% RSLogix 500 project Glycol_2.RSS, saved by version 12.00.00.00 %
PROJECT "GOODFOOD"    % processor: Bul.1763 MicroLogix 1100 Series B %

PROGRAM FILES
  LAD 2   24 rungs
  LAD 3   18 rungs
  LAD 4   25 rungs
  LAD 5   58 rungs

DATA FILES
  O0 OUTPUT  9 elements
  I1 INPUT  23 elements
  S2 STATUS  66 elements
  B3 BINARY  1 elements
  T4 TIMER  19 elements
  C5 COUNTER  9 elements
  R6 CONTROL  1 elements
  N7 INTEGER  11 elements
  F8 FLOAT  39 elements
  F9   45 elements
  B10   2 elements
  F11   14 elements
  F12   8 elements
  T13   7 elements
  F14   10 elements
  F15   10 elements
  B16   2 elements
  PD17   1 elements
  PD18   1 elements
  N19   23 elements
  F20   40 elements

LADDER 2
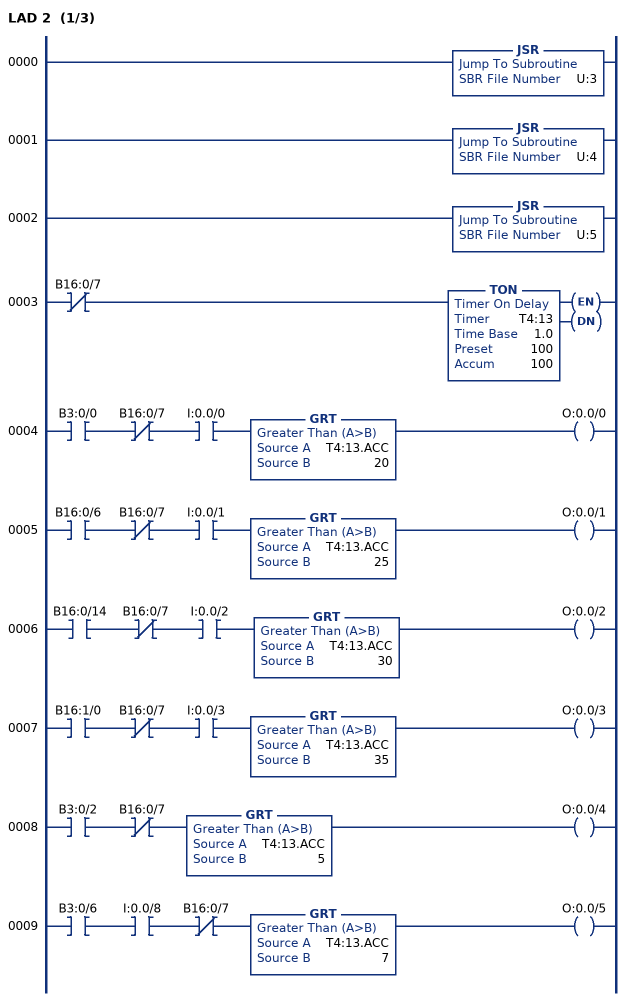
% Rung: 0 %
SOR JSR U:3 EOR
% Rung: 1 %
SOR JSR U:4 EOR
% Rung: 2 %
SOR JSR U:5 EOR
% Rung: 3 %
SOR XIO B16:0/7 TON T4:13 1.0 100 100 EOR
% Rung: 4 %
SOR XIC B3:0/0 XIO B16:0/7 XIC I:0.0/0 GRT T4:13.ACC 20 OTE O:0.0/0 EOR
% Rung: 5 %
SOR XIC B16:0/6 XIO B16:0/7 XIC I:0.0/1 GRT T4:13.ACC 25 OTE O:0.0/1 EOR
% Rung: 6 %
SOR XIC B16:0/14 XIO B16:0/7 XIC I:0.0/2 GRT T4:13.ACC 30 OTE O:0.0/2 EOR
% Rung: 7 %
SOR XIC B16:1/0 XIO B16:0/7 XIC I:0.0/3 GRT T4:13.ACC 35 OTE O:0.0/3 EOR
% Rung: 8 %
SOR XIC B3:0/2 XIO B16:0/7 GRT T4:13.ACC 5 OTE O:0.0/4 EOR
% Rung: 9 %
SOR XIC B3:0/6 XIC I:0.0/8 XIO B16:0/7 GRT T4:13.ACC 7 OTE O:0.0/5 EOR

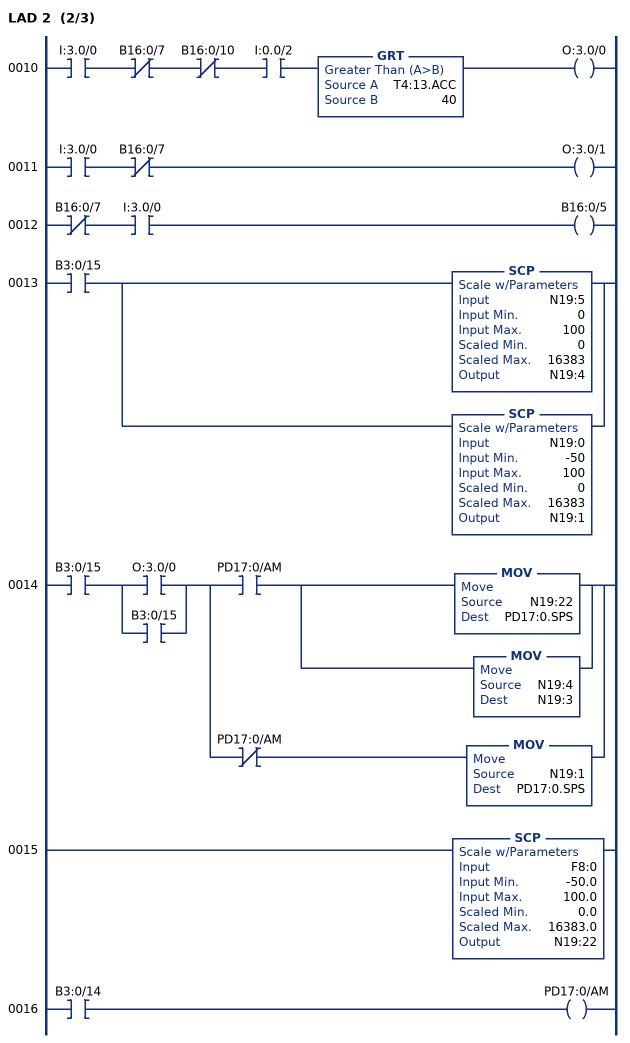
% Rung: 10 %
SOR XIC I:3.0/0 XIO B16:0/7 XIO B16:0/10 XIC I:0.0/2 GRT T4:13.ACC 40 OTE O:3.0/0 EOR
% Rung: 11 %
SOR XIC I:3.0/0 XIO B16:0/7 OTE O:3.0/1 EOR
% Rung: 12 %
SOR XIO B16:0/7 XIC I:3.0/0 OTE B16:0/5 EOR
% Rung: 13 %
SOR XIC B3:0/15 BST SCP N19:5 0 100 0 16383 N19:4 NXB SCP N19:0 -50 100 0 16383 N19:1 BND EOR
% Rung: 14 %
SOR XIC B3:0/15 BST XIC O:3.0/0 NXB XIC B3:0/15 BND BST XIC PD17:0/AM BST MOV N19:22 PD17:0.SPS NXB MOV N19:4 N19:3 BND NXB XIO PD17:0/AM MOV N19:1 PD17:0.SPS BND EOR
% Rung: 15 %
SOR SCP F8:0 -50.0 100.0 0.0 16383.0 N19:22 EOR
% Rung: 16 %
SOR XIC B3:0/14 OTE PD17:0/AM EOR

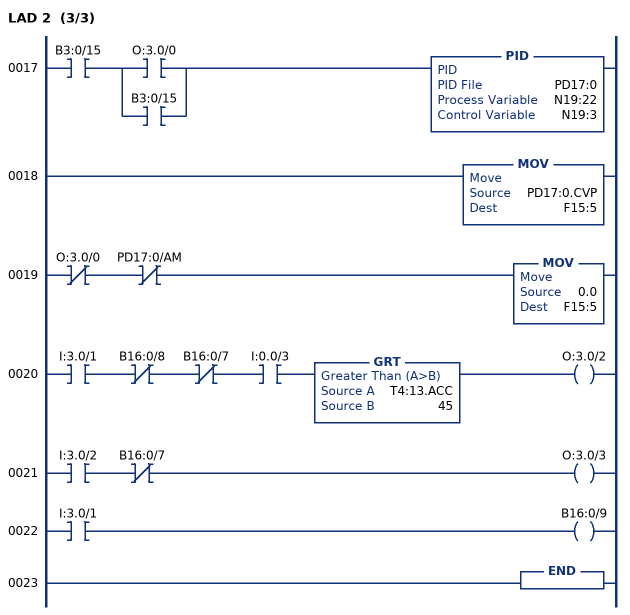
% Rung: 17 %
SOR XIC B3:0/15 BST XIC O:3.0/0 NXB XIC B3:0/15 BND PID PD17:0 N19:22 N19:3 EOR
% Rung: 18 %
SOR MOV PD17:0.CVP F15:5 EOR
% Rung: 19 %
SOR XIO O:3.0/0 XIO PD17:0/AM MOV 0.0 F15:5 EOR
% Rung: 20 %
SOR XIC I:3.0/1 XIO B16:0/8 XIO B16:0/7 XIC I:0.0/3 GRT T4:13.ACC 45 OTE O:3.0/2 EOR
% Rung: 21 %
SOR XIC I:3.0/2 XIO B16:0/7 OTE O:3.0/3 EOR
% Rung: 22 %
SOR XIC I:3.0/1 OTE B16:0/9 EOR
% Rung: 23 %
SOR END EOR

LADDER 3
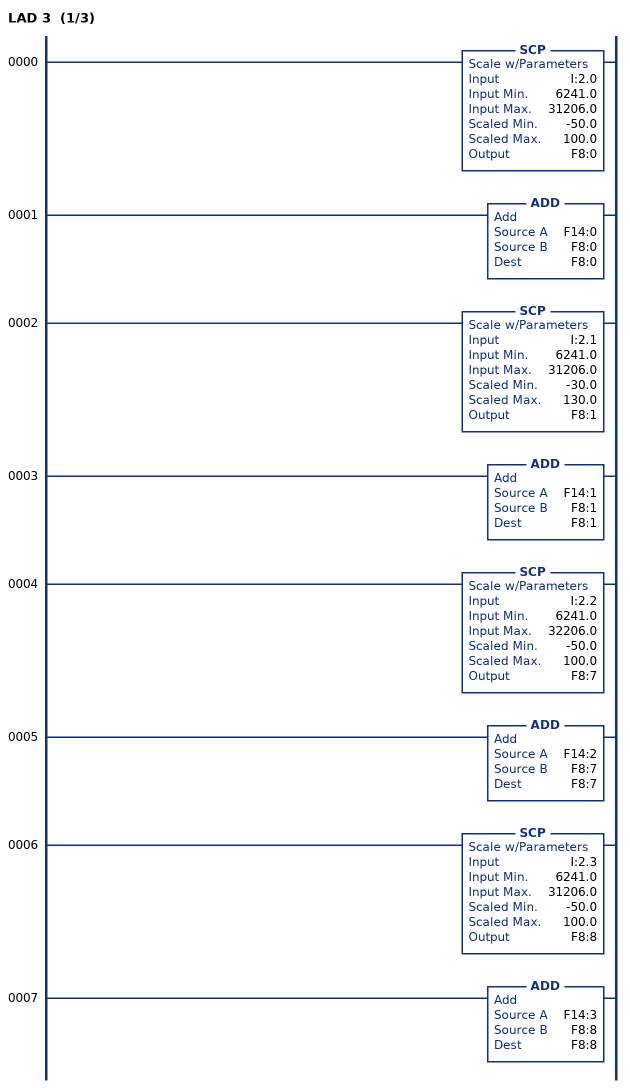
% Rung: 0 %
SOR SCP I:2.0 6241.0 31206.0 -50.0 100.0 F8:0 EOR
% Rung: 1 %
SOR ADD F14:0 F8:0 F8:0 EOR
% Rung: 2 %
SOR SCP I:2.1 6241.0 31206.0 -30.0 130.0 F8:1 EOR
% Rung: 3 %
SOR ADD F14:1 F8:1 F8:1 EOR
% Rung: 4 %
SOR SCP I:2.2 6241.0 32206.0 -50.0 100.0 F8:7 EOR
% Rung: 5 %
SOR ADD F14:2 F8:7 F8:7 EOR
% Rung: 6 %
SOR SCP I:2.3 6241.0 31206.0 -50.0 100.0 F8:8 EOR
% Rung: 7 %
SOR ADD F14:3 F8:8 F8:8 EOR

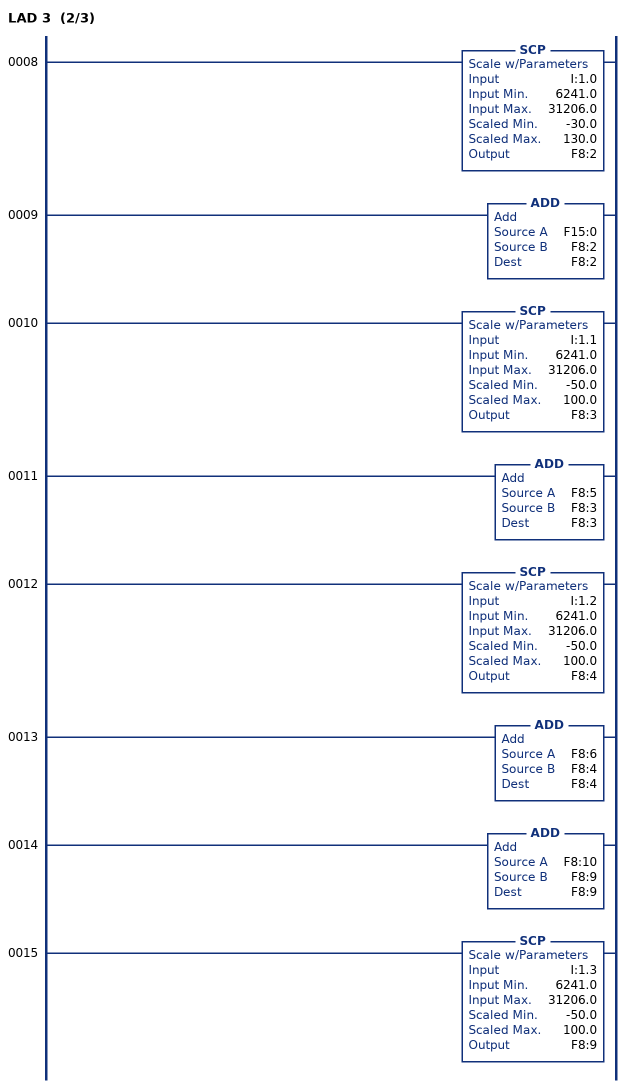
% Rung: 8 %
SOR SCP I:1.0 6241.0 31206.0 -30.0 130.0 F8:2 EOR
% Rung: 9 %
SOR ADD F15:0 F8:2 F8:2 EOR
% Rung: 10 %
SOR SCP I:1.1 6241.0 31206.0 -50.0 100.0 F8:3 EOR
% Rung: 11 %
SOR ADD F8:5 F8:3 F8:3 EOR
% Rung: 12 %
SOR SCP I:1.2 6241.0 31206.0 -50.0 100.0 F8:4 EOR
% Rung: 13 %
SOR ADD F8:6 F8:4 F8:4 EOR
% Rung: 14 %
SOR ADD F8:10 F8:9 F8:9 EOR
% Rung: 15 %
SOR SCP I:1.3 6241.0 31206.0 -50.0 100.0 F8:9 EOR

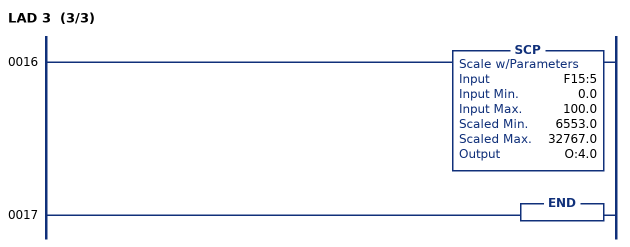
% Rung: 16 %
SOR SCP F15:5 0.0 100.0 6553.0 32767.0 O:4.0 EOR
% Rung: 17 %
SOR END EOR

LADDER 4
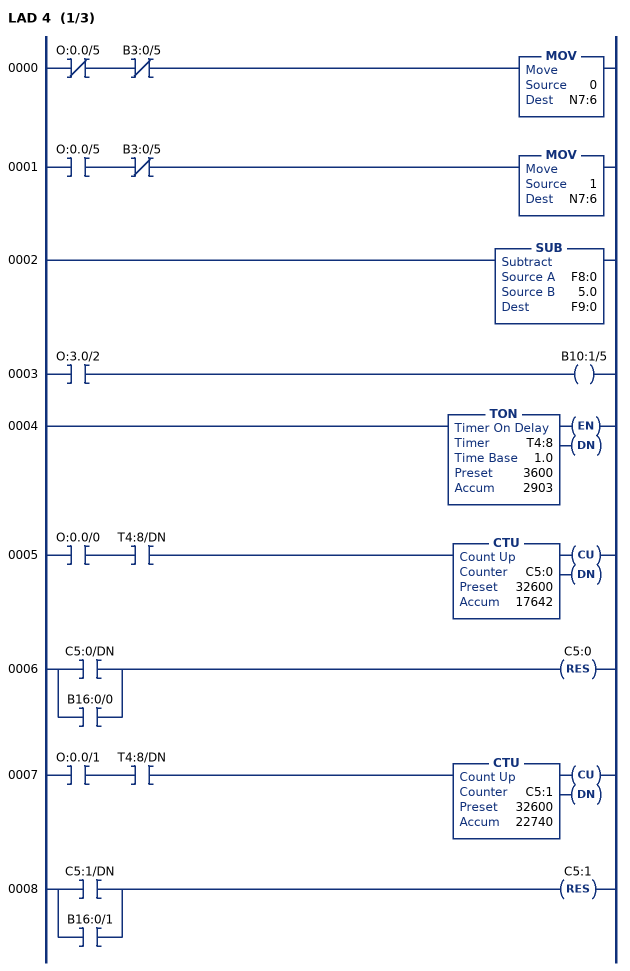
% Rung: 0 %
SOR XIO O:0.0/5 XIO B3:0/5 MOV 0 N7:6 EOR
% Rung: 1 %
SOR XIC O:0.0/5 XIO B3:0/5 MOV 1 N7:6 EOR
% Rung: 2 %
SOR SUB F8:0 5.0 F9:0 EOR
% Rung: 3 %
SOR XIC O:3.0/2 OTE B10:1/5 EOR
% Rung: 4 %
SOR TON T4:8 1.0 3600 2903 EOR
% Rung: 5 %
SOR XIC O:0.0/0 XIC T4:8/DN CTU C5:0 32600 17642 EOR
% Rung: 6 %
SOR BST XIC C5:0/DN NXB XIC B16:0/0 BND RES C5:0 EOR
% Rung: 7 %
SOR XIC O:0.0/1 XIC T4:8/DN CTU C5:1 32600 22740 EOR
% Rung: 8 %
SOR BST XIC C5:1/DN NXB XIC B16:0/1 BND RES C5:1 EOR

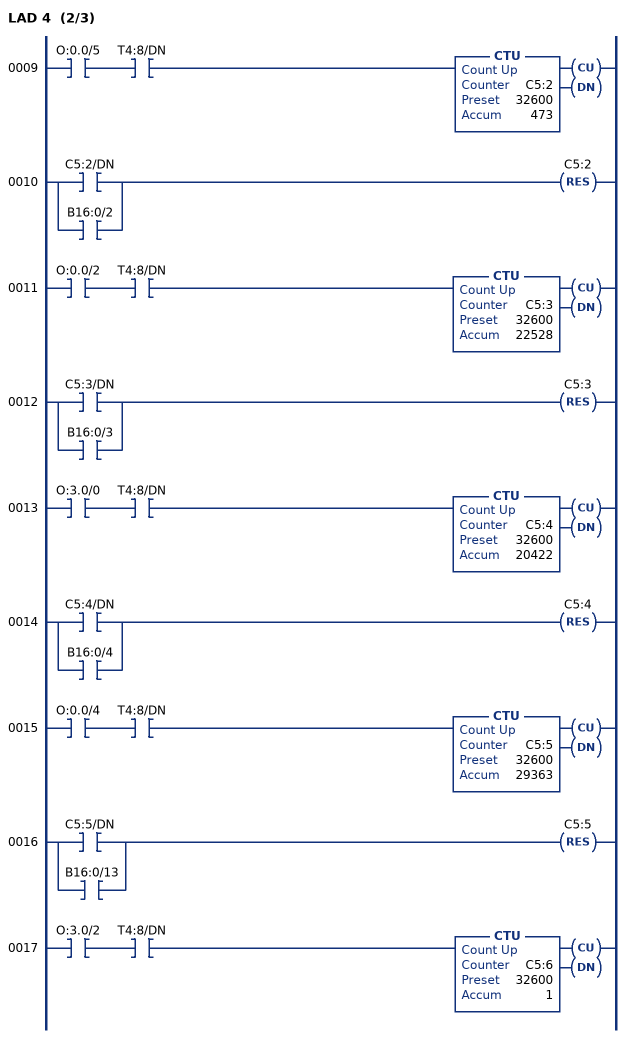
% Rung: 9 %
SOR XIC O:0.0/5 XIC T4:8/DN CTU C5:2 32600 473 EOR
% Rung: 10 %
SOR BST XIC C5:2/DN NXB XIC B16:0/2 BND RES C5:2 EOR
% Rung: 11 %
SOR XIC O:0.0/2 XIC T4:8/DN CTU C5:3 32600 22528 EOR
% Rung: 12 %
SOR BST XIC C5:3/DN NXB XIC B16:0/3 BND RES C5:3 EOR
% Rung: 13 %
SOR XIC O:3.0/0 XIC T4:8/DN CTU C5:4 32600 20422 EOR
% Rung: 14 %
SOR BST XIC C5:4/DN NXB XIC B16:0/4 BND RES C5:4 EOR
% Rung: 15 %
SOR XIC O:0.0/4 XIC T4:8/DN CTU C5:5 32600 29363 EOR
% Rung: 16 %
SOR BST XIC C5:5/DN NXB XIC B16:0/13 BND RES C5:5 EOR
% Rung: 17 %
SOR XIC O:3.0/2 XIC T4:8/DN CTU C5:6 32600 1 EOR

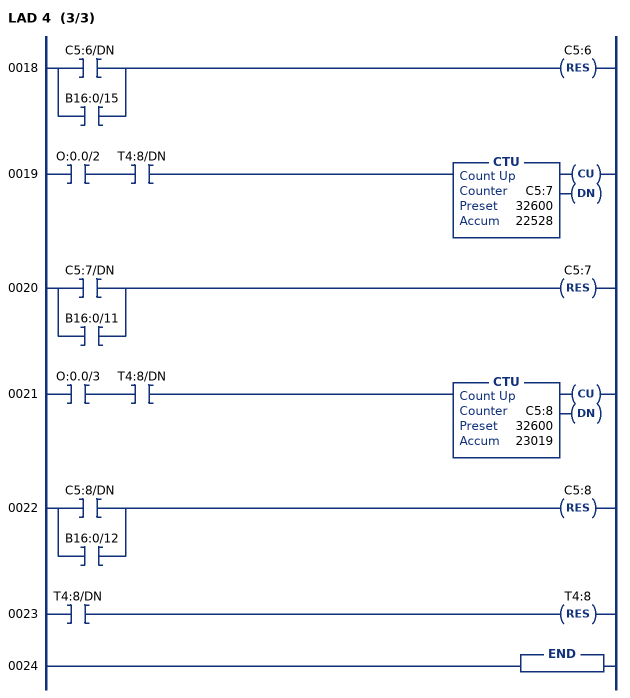
% Rung: 18 %
SOR BST XIC C5:6/DN NXB XIC B16:0/15 BND RES C5:6 EOR
% Rung: 19 %
SOR XIC O:0.0/2 XIC T4:8/DN CTU C5:7 32600 22528 EOR
% Rung: 20 %
SOR BST XIC C5:7/DN NXB XIC B16:0/11 BND RES C5:7 EOR
% Rung: 21 %
SOR XIC O:0.0/3 XIC T4:8/DN CTU C5:8 32600 23019 EOR
% Rung: 22 %
SOR BST XIC C5:8/DN NXB XIC B16:0/12 BND RES C5:8 EOR
% Rung: 23 %
SOR XIC T4:8/DN RES T4:8 EOR
% Rung: 24 %
SOR END EOR

LADDER 5
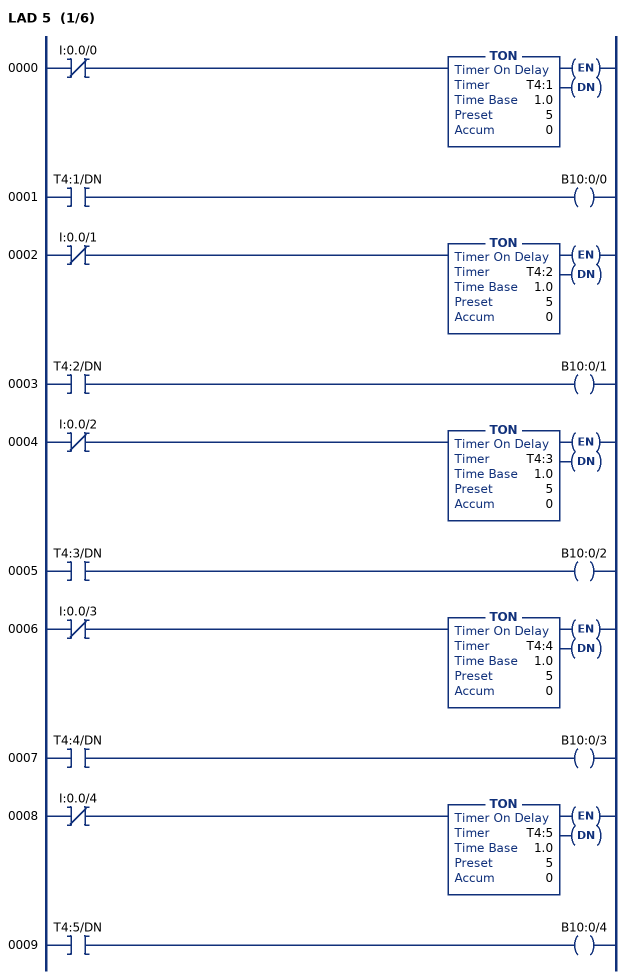
% Rung: 0 %
SOR XIO I:0.0/0 TON T4:1 1.0 5 0 EOR
% Rung: 1 %
SOR XIC T4:1/DN OTE B10:0/0 EOR
% Rung: 2 %
SOR XIO I:0.0/1 TON T4:2 1.0 5 0 EOR
% Rung: 3 %
SOR XIC T4:2/DN OTE B10:0/1 EOR
% Rung: 4 %
SOR XIO I:0.0/2 TON T4:3 1.0 5 0 EOR
% Rung: 5 %
SOR XIC T4:3/DN OTE B10:0/2 EOR
% Rung: 6 %
SOR XIO I:0.0/3 TON T4:4 1.0 5 0 EOR
% Rung: 7 %
SOR XIC T4:4/DN OTE B10:0/3 EOR
% Rung: 8 %
SOR XIO I:0.0/4 TON T4:5 1.0 5 0 EOR
% Rung: 9 %
SOR XIC T4:5/DN OTE B10:0/4 EOR

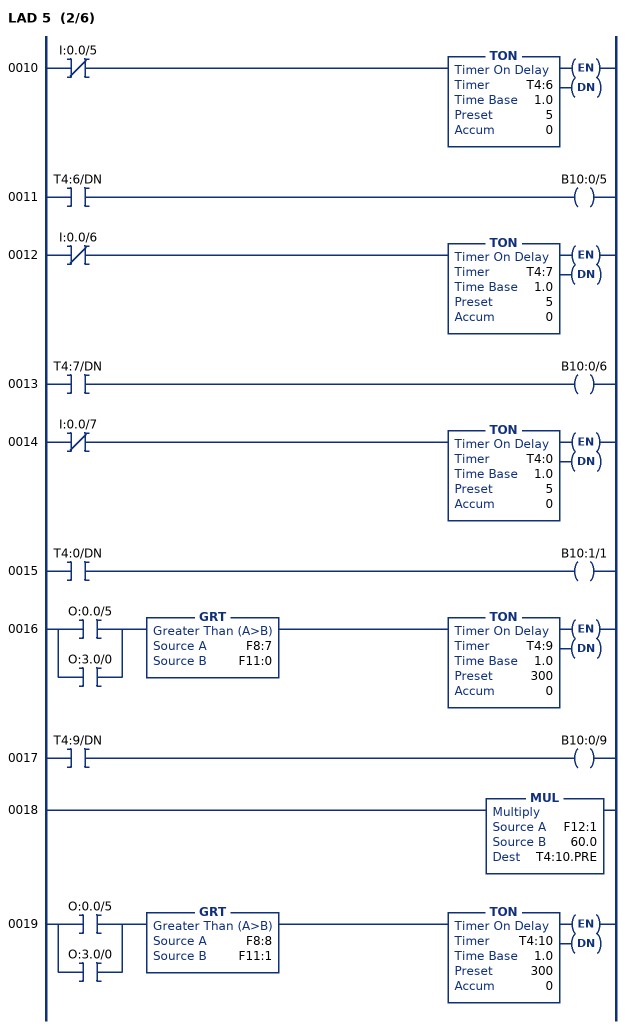
% Rung: 10 %
SOR XIO I:0.0/5 TON T4:6 1.0 5 0 EOR
% Rung: 11 %
SOR XIC T4:6/DN OTE B10:0/5 EOR
% Rung: 12 %
SOR XIO I:0.0/6 TON T4:7 1.0 5 0 EOR
% Rung: 13 %
SOR XIC T4:7/DN OTE B10:0/6 EOR
% Rung: 14 %
SOR XIO I:0.0/7 TON T4:0 1.0 5 0 EOR
% Rung: 15 %
SOR XIC T4:0/DN OTE B10:1/1 EOR
% Rung: 16 %
SOR BST XIC O:0.0/5 NXB XIC O:3.0/0 BND GRT F8:7 F11:0 TON T4:9 1.0 300 0 EOR
% Rung: 17 %
SOR XIC T4:9/DN OTE B10:0/9 EOR
% Rung: 18 %
SOR MUL F12:1 60.0 T4:10.PRE EOR
% Rung: 19 %
SOR BST XIC O:0.0/5 NXB XIC O:3.0/0 BND GRT F8:8 F11:1 TON T4:10 1.0 300 0 EOR

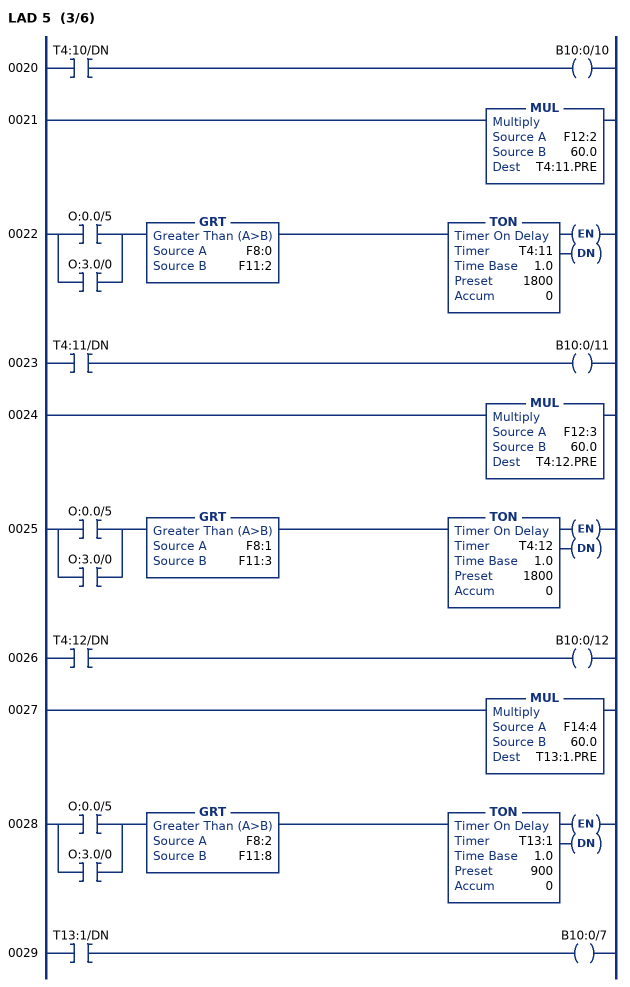
% Rung: 20 %
SOR XIC T4:10/DN OTE B10:0/10 EOR
% Rung: 21 %
SOR MUL F12:2 60.0 T4:11.PRE EOR
% Rung: 22 %
SOR BST XIC O:0.0/5 NXB XIC O:3.0/0 BND GRT F8:0 F11:2 TON T4:11 1.0 1800 0 EOR
% Rung: 23 %
SOR XIC T4:11/DN OTE B10:0/11 EOR
% Rung: 24 %
SOR MUL F12:3 60.0 T4:12.PRE EOR
% Rung: 25 %
SOR BST XIC O:0.0/5 NXB XIC O:3.0/0 BND GRT F8:1 F11:3 TON T4:12 1.0 1800 0 EOR
% Rung: 26 %
SOR XIC T4:12/DN OTE B10:0/12 EOR
% Rung: 27 %
SOR MUL F14:4 60.0 T13:1.PRE EOR
% Rung: 28 %
SOR BST XIC O:0.0/5 NXB XIC O:3.0/0 BND GRT F8:2 F11:8 TON T13:1 1.0 900 0 EOR
% Rung: 29 %
SOR XIC T13:1/DN OTE B10:0/7 EOR

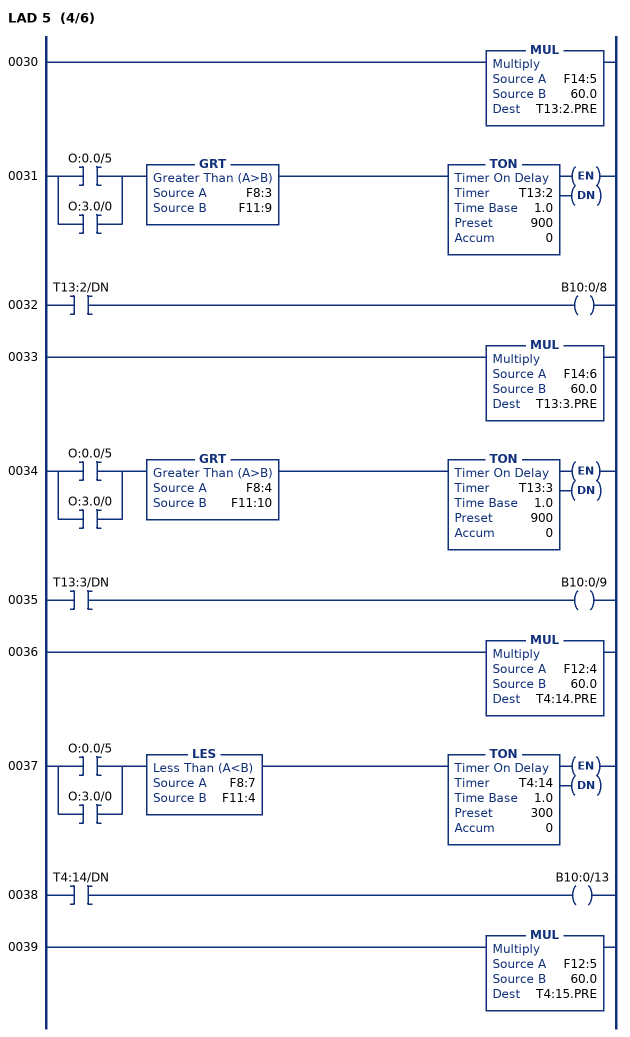
% Rung: 30 %
SOR MUL F14:5 60.0 T13:2.PRE EOR
% Rung: 31 %
SOR BST XIC O:0.0/5 NXB XIC O:3.0/0 BND GRT F8:3 F11:9 TON T13:2 1.0 900 0 EOR
% Rung: 32 %
SOR XIC T13:2/DN OTE B10:0/8 EOR
% Rung: 33 %
SOR MUL F14:6 60.0 T13:3.PRE EOR
% Rung: 34 %
SOR BST XIC O:0.0/5 NXB XIC O:3.0/0 BND GRT F8:4 F11:10 TON T13:3 1.0 900 0 EOR
% Rung: 35 %
SOR XIC T13:3/DN OTE B10:0/9 EOR
% Rung: 36 %
SOR MUL F12:4 60.0 T4:14.PRE EOR
% Rung: 37 %
SOR BST XIC O:0.0/5 NXB XIC O:3.0/0 BND LES F8:7 F11:4 TON T4:14 1.0 300 0 EOR
% Rung: 38 %
SOR XIC T4:14/DN OTE B10:0/13 EOR
% Rung: 39 %
SOR MUL F12:5 60.0 T4:15.PRE EOR

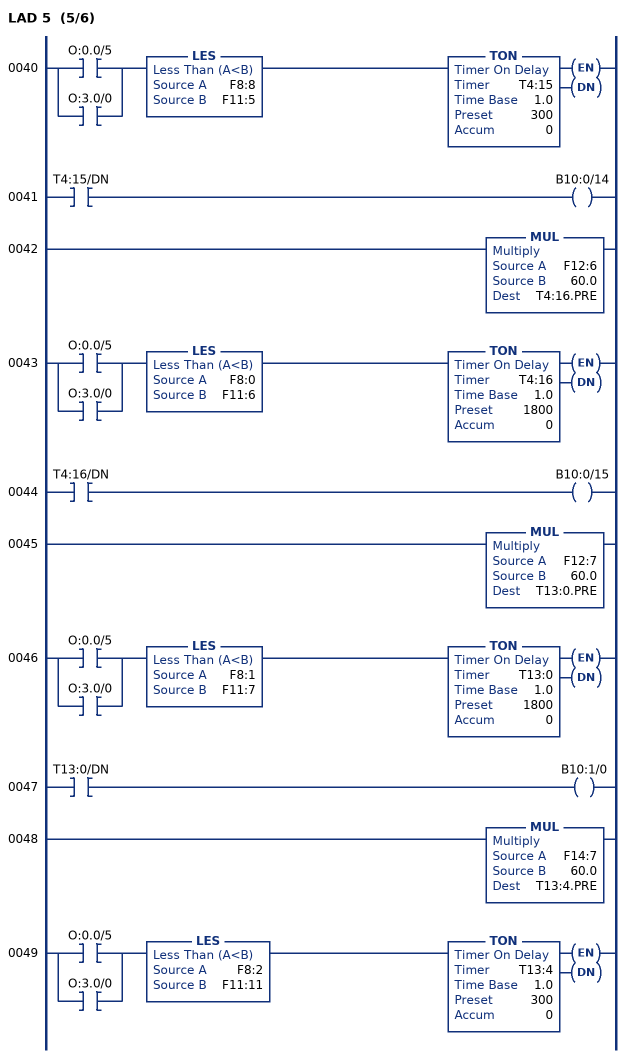
% Rung: 40 %
SOR BST XIC O:0.0/5 NXB XIC O:3.0/0 BND LES F8:8 F11:5 TON T4:15 1.0 300 0 EOR
% Rung: 41 %
SOR XIC T4:15/DN OTE B10:0/14 EOR
% Rung: 42 %
SOR MUL F12:6 60.0 T4:16.PRE EOR
% Rung: 43 %
SOR BST XIC O:0.0/5 NXB XIC O:3.0/0 BND LES F8:0 F11:6 TON T4:16 1.0 1800 0 EOR
% Rung: 44 %
SOR XIC T4:16/DN OTE B10:0/15 EOR
% Rung: 45 %
SOR MUL F12:7 60.0 T13:0.PRE EOR
% Rung: 46 %
SOR BST XIC O:0.0/5 NXB XIC O:3.0/0 BND LES F8:1 F11:7 TON T13:0 1.0 1800 0 EOR
% Rung: 47 %
SOR XIC T13:0/DN OTE B10:1/0 EOR
% Rung: 48 %
SOR MUL F14:7 60.0 T13:4.PRE EOR
% Rung: 49 %
SOR BST XIC O:0.0/5 NXB XIC O:3.0/0 BND LES F8:2 F11:11 TON T13:4 1.0 300 0 EOR

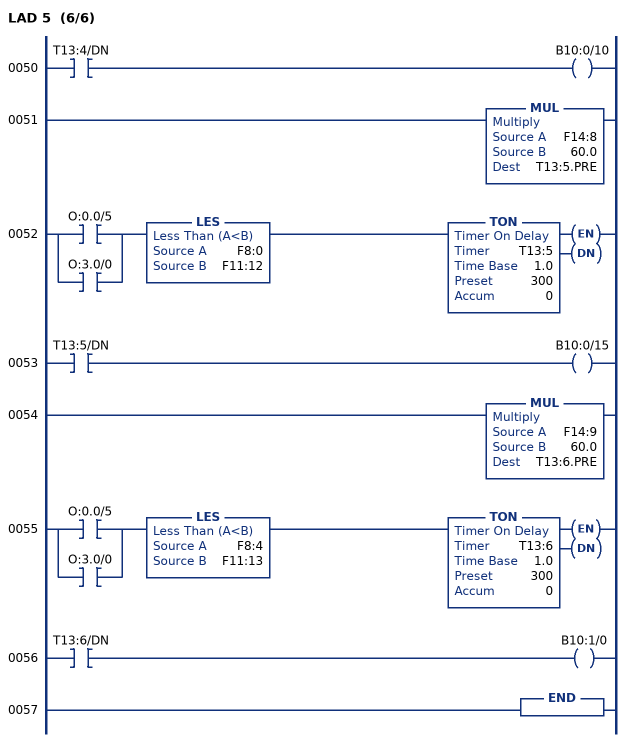
% Rung: 50 %
SOR XIC T13:4/DN OTE B10:0/10 EOR
% Rung: 51 %
SOR MUL F14:8 60.0 T13:5.PRE EOR
% Rung: 52 %
SOR BST XIC O:0.0/5 NXB XIC O:3.0/0 BND LES F8:0 F11:12 TON T13:5 1.0 300 0 EOR
% Rung: 53 %
SOR XIC T13:5/DN OTE B10:0/15 EOR
% Rung: 54 %
SOR MUL F14:9 60.0 T13:6.PRE EOR
% Rung: 55 %
SOR BST XIC O:0.0/5 NXB XIC O:3.0/0 BND LES F8:4 F11:13 TON T13:6 1.0 300 0 EOR
% Rung: 56 %
SOR XIC T13:6/DN OTE B10:1/0 EOR
% Rung: 57 %
SOR END EOR

DATA TABLE (non-zero values as saved)
DATA B3
% B3:0 % 0X80C7
DATA T4
% .PRE .ACC %
% T4:0 % 5 0
% T4:1 % 5 0
% T4:2 % 5 0
% T4:3 % 5 0
% T4:4 % 5 0
% T4:5 % 5 0
% T4:6 % 5 0
% T4:7 % 5 0
% T4:8 % 3600 2903
% T4:9 % 300 0
% T4:10 % 300 0
% T4:11 % 1800 0
% T4:12 % 1800 0
% T4:13 % 100 100
% T4:14 % 300 0
% T4:15 % 300 0
% T4:16 % 1800 0
% T4:17 % 5 0
% T4:18 % 5 0
DATA C5
% .PRE .ACC %
% C5:0 % 32600 17642
% C5:1 % 32600 22740
% C5:2 % 32600 473
% C5:3 % 32600 22528
% C5:4 % 32600 20422
% C5:5 % 32600 29363
% C5:6 % 32600 1
% C5:7 % 32600 22528
% C5:8 % 32600 23019
DATA N7
% N7:0 % 0 1 2 75 10976 0 1 0 0 0
DATA F8
% F8:0 % 40.75706 34.81394 37.47713 -89.36846 29.82175
% F8:5 % -1.9 0 35.38538 35.15239 27.857
% F8:10 % 34.52032 0 0 0 0
DATA F9
% F9:0 % 35.75706 0 0 0 0
DATA F11
% F11:0 % 60 60 45 45 20
% F11:5 % 20 15 15 60 60
% F11:10 % 60 25 25 25
DATA F12
% F12:0 % 5 5 30 30 5
% F12:5 % 5 30 30
DATA T13
% .PRE .ACC %
% T13:0 % 1800 0
% T13:1 % 900 0
% T13:2 % 900 0
% T13:3 % 900 0
% T13:4 % 300 0
% T13:5 % 300 0
% T13:6 % 300 0
DATA F14
% F14:0 % 0 0 -0.9 -3.7 15
% F14:5 % 15 15 5 5 5
DATA F15
% F15:0 % -1.9 0 0 0 0
DATA B16
% B16:0 % 0X4160 0X0001
DATA N19
% N19:0 % 25 8192 415 0 4915 30 0 0 0 0
% N19:20 % 0 41 9914
